(* PLC project x, CODESYS CODESYS V3.5 SP11 *)
(* stored: creationDateTime 2026-08-04T14:40:27 *)

PROGRAM LD_PAR
  VAR
    xA : BOOL;
  END_VAR

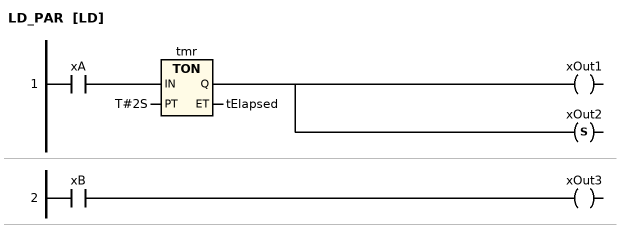
(* LD diagram, written out as Structured Text *)
(* Network one comment *)
tmr(IN := xA, PT := T#2S);
xOut1 := tmr.Q;
IF tmr.Q THEN xOut2 := TRUE; END_IF;
tElapsed := tmr.ET;
(* Network two comment *)
xOut3 := xB;
END_PROGRAM
